(* IEC 61131-3 sources: Lasal/CPU_5344_V01/Class/Logic_Or_2, 1 file *)

(* ---- Logic_Or_2.st ---- *)
(*!
<Class
	Name               = "Logic_Or_2"
	Revision           = "1.1"
	RealtimeTask       = "false"
	CyclicTask         = "false"
	BackgroundTask     = "false"
	Sigmatek           = "true"
	OSInterface        = "false"
	HighPriority       = "false"
	Automatic          = "false"
	UpdateMode         = "Prescan"
	IconPath           = ".\Class\Logic_Or_2\Logic_Or_Base.ico"
	SharedCommandTable = "true"
	Objectsize         = "(284,120)"
	Comment            = "V1.1 Logic OR class with 2 operands">
	<Channels>
		<Server
			Name           = "Result"
			Initialize     = "false"
			Visualized     = "true"
			WriteProtected = "true"
			Comment        = "result of logic operation">
		</Server>
		<Client Name="Op1" Required="false" Internal="false" Comment="Operand 1"/>
		<Client Name="Op2" Required="false" Internal="false" Comment="Operand 2"/>
	</Channels>
	<Network Name="Logic_Or_2">
		<!-- List of Components in this network -->
		<Components>
			<Object
				Name       = "_base"
				Class      = "Logic_Or_Base"
				Position   = "(570,1110)"
				Visualized = "true">
				<Channels>
					<Server Name="Result"/>
				</Channels>
			</Object>
		</Components>
		<Comments>
		</Comments>
		<!-- List of Connections in this network -->
		<Connections>
			<Connection Source="this.Result" Destination="_base.Result" Vertices="(1042,210),(870,1200),"/>
		</Connections>
		<!-- Headerfiles -->
		<Options>
		</Options>
	</Network>
</Class>
*)
#pragma using Logic_Or_Base

Logic_Or_2 : CLASS
: Logic_Or_Base
  //Servers:
  //Clients:
	Op1 	: CltCh_DINT;
	Op2 	: CltCh_DINT;
  //Variables:
  //Functions:
  //Tables:
	FUNCTION @STD
		VAR_OUTPUT
			ret_code	: CONFSTATES;
		END_VAR;
	FUNCTION GLOBAL TAB @CT_;
END_CLASS;
